INTERFACE I_Subscriber

METHOD Update : BOOL
VAR_INPUT
	Value : LREAL;
END_VAR
END_METHOD

END_INTERFACE

(* stored: Version 1.1.0.1, ProductVersion 3.1.4022.18
   Itf I_Subscriber: Id {f9510eea-3e34-4d2b-894c-a5b9af453fe1}
   Method Update: Id {427e1344-07e1-4750-bd9a-bd231d31baea} *)
